{attribute addProperty BoxType "KL8001-0002"}
{attribute addProperty Id "State_0AT %I*USINT000Data_In_0AT %I*UINT000State_ExtAT %I*USINT000Ctrl_0AT %Q*USINT000Data_Out_0AT %Q*UINT000Ctrl_ExtAT %Q*USINT000"}
{attribute addProperty CRC "490576518"}
{attribute addProperty SizeInBites "0"}
{attribute addProperty SizeInBytes "0"}
TYPE Channel_1D3D9A86 :
STRUCT
	{attribute addProperty Name "State_0"}
	State_0 AT %I* : USINT;
	{attribute addProperty Name "Data_In_0"}
	Data_In_0 AT %I* : UINT;
	{attribute addProperty Name "State_Ext"}
	State_Ext AT %I* : USINT;
	{attribute addProperty Name "Ctrl_0"}
	Ctrl_0 AT %Q* : USINT;
	{attribute addProperty Name "Data_Out_0"}
	Data_Out_0 AT %Q* : UINT;
	{attribute addProperty Name "Ctrl_Ext"}
	Ctrl_Ext AT %Q* : USINT;
END_STRUCT
END_TYPE

(* stored: Version 1.2.0.0, ProductVersion 3.1.4024.9
   DUT Channel_1D3D9A86: Id {48861b15-fbac-45d5-8502-a85d5e3f8d35} *)
